//-----------------------------------------------------------------------------------------
//
//                  				ST_Alarm
//
//								Variables alarme			
//-----------------------------------------------------------------------------------------
//
//Auteur: G.GOETZ (inspired by S.MANTZER)
//Création: 21.01.2026
//Dernière modification : 21.01.2026 (G.GOETZ)
//       			
//-----------------------------------------------------------------------------------------
//
//     							Liste des modifications  	
//
// 21.01.2026 (G.GOETZ) -> Création		
//-----------------------------------------------------------------------------------------

TYPE ST_Alarm :
STRUCT
	
	(** FB **)
	fbAlarm : FB_TcAlarm;

END_STRUCT
END_TYPE

(* stored: Version 1.1.0.1, ProductVersion 3.1.4024.13
   DUT ST_Alarm: Id {ac78ce84-daea-4748-a48d-6b1bf6c21ed8} *)
